  994 = 'S3_Prompts Default 994' | German: 'S3_Prompts German 994' | French: 'S3_Prompts French 994'
  995 = 'S3_Prompts Default 995' | German: 'S3_Prompts German 995' | French: 'S3_Prompts French 995'
  996 = 'S3_Prompts Default 996' | German: 'S3_Prompts German 996' | French: 'S3_Prompts French 996'
  997 = 'S3_Prompts Default 997' | German: 'S3_Prompts German 997' | French: 'S3_Prompts French 997'
  998 = 'S3_Prompts Default 998' | German: 'S3_Prompts German 998' | French: 'S3_Prompts French 998'
  999 = 'S3_Prompts Default 999' | German: 'S3_Prompts German 999' | French: 'S3_Prompts French 999'
  1000 = 'S3_Prompts Default 1000' | German: 'S3_Prompts German 1000' | French: 'S3_Prompts French 1000'
   = ''
END_TEXTLIST

(* stored: Version 1.1.0.1, ProductVersion 3.1.4024.12
   TextList S3_Prompts: Id {f91ea3fe-05c5-4791-81a6-65e12d9c4dcd} *)
